// TIA Portal V20 export
DATA_BLOCK "IDB_ManualControl"   // DB50
// stored: InstanceOfName Global.FB_ManualControl, InstanceOfType FB, Namespace Global
"Global.FB_ManualControl"
   // VAR RETAIN
   //    "Counter" { S7_SetPoint := 'True'} : CTU_INT;
   // END_VAR
BEGIN
END_DATA_BLOCK
